// TIA Portal V16 export
// export: Created 2024-03-27T10:04:39.8939168Z, ExportSetting WithDefaults, DisplayName Totally Integrated Automation Portal, DisplayVersion V16, DisplayName TIA Portal Version Control Interface, DisplayVersion V16, DisplayName TIA Portal Openness, DisplayVersion V16, DisplayName STEP 7 Professional, DisplayVersion V16, DisplayName STEP 7 Safety, DisplayVersion V16, DisplayName WinCC Advanced, DisplayVersion V16
TYPE "UR_T2O"
// stored: IsFailsafeCompliant false
   STRUCT
      State { ExternalAccessible := 'False'; ExternalVisible := 'False'; ExternalWritable := 'False'; S7_SetPoint := 'True'} : "UR_1_T2O_State";
      IO { S7_SetPoint := 'True'} : "UR_2_T2O_IO";
      Joints { S7_SetPoint := 'True'} : "UR_3_T2O_Joints";
      TCP { S7_SetPoint := 'True'} : "UR_4_T2O_TCP";
      Bits { S7_SetPoint := 'True'} : "UR_5_T2O_BitRegisters";
      Ints { S7_SetPoint := 'True'} : "UR_6_T2O_IntRegisters";
      Floats { S7_SetPoint := 'True'} : "UR_7_T2O_FloatRegisters";
   END_STRUCT;
END_TYPE
